{attribute wpf [Container(Layout.UniformGrid)]}
TYPE UniformGridLayout:
STRUCT
	_various_types: VariousTypes;
END_STRUCT
END_TYPE

(* stored: Version 1.1.0.1, ProductVersion 3.1.4024.9
   DUT UniformGridLayout: Id {6cccbacb-de95-4d2f-83ae-54edf4bba15d} *)
